Staubli VAL3: StaubliUI.pjx

--- StaubliUI.pjx ---
Parameters version=s7.7 stackSize=15000 millimeterUnit=true
Program file=Bool_Edit.pgx
Program file=BoolMess_Edit.pgx
Program file=Control_Action.pgx
Program file=Control_AxisPar.pgx
Program file=Control_BatPara.pgx
Program file=Control_BatPrt.pgx
Program file=Control_BatSpd.pgx
Program file=Control_Bottom.pgx
Program file=Control_BottomS.pgx
Program file=Control_CPreset.pgx
Program file=Control_Joint.pgx
Program file=Control_Lable.pgx
Program file=Control_Left.pgx
Program file=Control_LeftCut.pgx
Program file=Control_LeftS.pgx
Program file=Control_List.pgx
Program file=Control_List1S.pgx
Program file=Control_ListBS.pgx
Program file=Control_ListCls.pgx
Program file=Control_ListMC.pgx
Program file=Control_ListMCD.pgx
Program file=Control_ListS.pgx
Program file=Control_Loffset.pgx
Program file=Control_MCShow.pgx
Program file=Control_Mess.pgx
Program file=Control_Panel.pgx
Program file=Control_PanelB.pgx
Program file=Control_PanelD.pgx
Program file=Control_PanelMd.pgx
Program file=Control_PanelS.pgx
Program file=Control_PanelXY.pgx
Program file=Control_PanTitl.pgx
Program file=Control_Para.pgx
Program file=Control_Para1.pgx
Program file=Control_PatMove.pgx
Program file=Control_Point.pgx
Program file=Control_Preset.pgx
Program file=Control_Recipe.pgx
Program file=Control_Remote.pgx
Program file=Control_Scara.pgx
Program file=Control_Timer.pgx
Program file=Control_Traj.pgx
Program file=Control_YesNO.pgx
Program file=Float_Edit.pgx
Program file=Form_4jHome.pgx
Program file=Form_6jHome.pgx
Program file=Form_Action.pgx
Program file=Form_Bye.pgx
Program file=Form_Config.pgx
Program file=Form_LabelList.pgx
Program file=Form_Main.pgx
Program file=Form_MainS.pgx
Program file=Form_Panel.pgx
Program file=Form_Panel4P.pgx
Program file=Form_PanelBool.pgx
Program file=Form_PanelJoint.pgx
Program file=Form_PanelList.pgx
Program file=Form_PanelPoint.pgx
Program file=Form_PanelStr.pgx
Program file=Form_Patten.pgx
Program file=Form_PattenD.pgx
Program file=Form_PattenS.pgx
Program file=Form_Product.pgx
Program file=Form_ScaraRobot.pgx
Program file=Form_SelSharp.pgx
Program file=Form_SimArray.pgx
Program file=Form_Simulation.pgx
Program file=Form_Welcome.pgx
Program file=Int_Edit.pgx
Program file=Int_EditMin.pgx
Program file=Int_EditS.pgx
Program file=Key_ListBase.pgx
Program file=Key_ListMC.pgx
Program file=ReadMe.pgx
Program file=Sel_Edit.pgx
Program file=start.pgx
Program file=stop.pgx
Program file=Str_Edit.pgx
Program file=Str_SplitChar.pgx
Program file=Str_SplitComma.pgx
Data file=StaubliUI.dtx

--- Control_Action.pgx ---
public program Control_Action(num& x_nAction[] (dimensions=3), num x_nIndex, string& x_sIoName[], bool& x_bDigtal[])
  local string l_sItem[2]
  local num l_nNum
  local num l_nKey
  local num l_nData[24]
  local num l_nSelectIndex
  local bool l_bRes
  local num l_nBuff
begin
  //为LasMAN3.6 Action配置


  for l_nNum=0 to 11
    l_nData[l_nNum*2+0]=x_nAction[x_nIndex,l_nNum,0]
    l_nData[l_nNum*2+1]=x_nAction[x_nIndex,l_nNum,1]
  endFor
  l_sItem[0]="关"
  l_sItem[1]="开"

  resize(sBuff,1,24)


  call Control_BottomS("置空,清空,延时,插入,删除,,取消,确定")
  call Control_PanelXY(4,0,20,10)
  call Control_Panel("动作值")
  for l_nNum=0 to 11


    sBuff[l_nNum*2+0]=toString("",l_nNum+1)+"名称:"+x_sIoName[l_nData[l_nNum*2+0]]
    if x_bDigtal[l_nData[l_nNum*2]]
      sBuff[l_nNum*2+1]="值 : "+ l_sItem[sel(l_nData[l_nNum*2+1]==0,0,1)]
    else
      sBuff[l_nNum*2+1]="值 : "+toString(".1",l_nData[l_nNum*2+1])
    endIf

  endFor
  call Control_List(sBuff,l_nSelectIndex)


  //**********************************
  //按键响应
  while true
    l_nKey=getKey()

    switch l_nKey
      //向上
      case 261
        l_nSelectIndex=max(0,l_nSelectIndex-1)
      break

      //向下
      case 266
        l_nSelectIndex=min(l_nSelectIndex+1,23)
      break

      //编辑
      case 270
        if l_nSelectIndex%2==1
          if ! x_bDigtal[l_nData[l_nSelectIndex-1]]
            call Float_Edit(l_nData[l_nSelectIndex],nPanelLTopX+6,l_nSelectIndex+nPanelLTopY+1)
          else
            l_nData[l_nSelectIndex]=sel(l_nData[l_nSelectIndex]==1,1,0)
            call Sel_Edit(l_nData[l_nSelectIndex],nPanelLTopX+6,l_nSelectIndex+nPanelLTopY+1,l_sItem)
            l_nData[l_nSelectIndex]=sel(l_nData[l_nSelectIndex]==1,1,0)
          endIf

        else
          call Sel_Edit(l_nData[l_nSelectIndex],nPanelLTopX+7,l_nSelectIndex+nPanelLTopY+1,x_sIoName)
        endIf

      break

      case 271
        call Control_YesNO("确定设置为无IO信号吗?",l_bRes)
        if l_bRes

          l_nData[sel(l_nSelectIndex%2==0,l_nSelectIndex,l_nSelectIndex-1)]=0

        endIf

      break


      //全部置空
      case 272
        call Control_YesNO("确定全部清空吗?",l_bRes)
        if l_bRes
          for l_nNum=0 to 23
            l_nData[l_nNum]=0
          endFor


        endIf
      break


      case 273
        call Control_YesNO("确定要设置为延时吗?",l_bRes)
        if l_bRes
          l_nData[sel(l_nSelectIndex%2==0,l_nSelectIndex,l_nSelectIndex-1)]=165

        endIf
      break

      //插入
      case 274
        call Control_YesNO("确定要插入吗?",l_bRes)
        l_nBuff=roundDown(l_nSelectIndex/2)
        if l_bRes
          for l_nNum=23 to l_nBuff*2+2  step -1
            l_nData[l_nNum]=l_nData[l_nNum-2]
          endFor
          l_nData[l_nBuff*2]=l_nData[l_nBuff*2+1]=0

        endIf
      break


      //删除
      case 275
        call Control_YesNO("确定要删除吗?",l_bRes)
        l_nBuff=roundDown(l_nSelectIndex/2)
        if l_bRes
          for l_nNum=l_nBuff*2 to 21
            l_nData[l_nNum]=l_nData[l_nNum+2]
          endFor
          l_nData[23]=l_nData[22]=0

        endIf
      break





      //退出
      case 277
        cls()
        return

      break



      //取消
      case 278
        for l_nNum=0 to 11
          x_nAction[x_nIndex,l_nNum,0]= l_nData[l_nNum*2+0]
          x_nAction[x_nIndex,l_nNum,1]=l_nData[l_nNum*2+1]
        endFor
        return
      break

    endSwitch

    if l_nKey!=-1

      for l_nNum=0 to 11
        sBuff[l_nNum*2+0]=toString("",l_nNum+1)+"名称:"+x_sIoName[l_nData[l_nNum*2+0]]
        if x_bDigtal[l_nData[l_nNum*2]]
          sBuff[l_nNum*2+1]="值 : "+ l_sItem[sel(l_nData[l_nNum*2+1]==0,0,1)]
        else
          sBuff[l_nNum*2+1]="值 : "+toString(".2",l_nData[l_nNum*2+1])
        endIf

      endFor

      call Control_PanelXY(4,0,20,10)
      call Control_Panel("动作值")
      call Control_List(sBuff,l_nSelectIndex)
      call Control_BottomS("置空,清空,延时,插入,删除,,取消,确定")
    endIf


  endWhile





end

--- Control_AxisPar.pgx ---
public program Control_AxisPar(num& x_nPos, num& x_nSpeed, num& x_nPrecent, num& x_nJogSpeed, bool x_bTraj)
  local string l_sItem[6]
  local num l_nNum
  local num l_nKey
  local num l_nData[6]
  local num l_nSelectIndex
begin
  //为LasMAN3.6进行配置
  //修改点位的参数


  //通过局部变量来实现内部存储


  l_nData[0]=x_nPos
  l_nData[1]=x_nSpeed
  l_nData[2]=x_nPrecent
  l_nData[3]=x_nJogSpeed

  l_sItem[0]="位置mm   :"+toString(".3",l_nData[0])
  l_sItem[1]="速度m/min:"+toString(".3",l_nData[1])
  l_sItem[2]="比例分度 :"+toString(".3",l_nData[2])
  l_sItem[3]="点动速度 :"+toString(".3",l_nData[3])
  call Control_BottomS(",,,,,,取消,确定")

  call Control_PanelXY(8,0,17,4)
  call Control_Panel("参数")
  call Control_List(l_sItem,l_nSelectIndex)


  //按键响应
  while true
    l_nKey=getKey()

    switch l_nKey
      case 261
        l_nSelectIndex=max(0,l_nSelectIndex-1)
      break

      case 266
        if x_bTraj
          l_nSelectIndex=min(1,l_nSelectIndex+1)
        else
           l_nSelectIndex=min(3,l_nSelectIndex+1)
        endIf

      break

      case 278

        x_nPos=l_nData[0]
        x_nSpeed=l_nData[1]
        x_nPrecent=l_nData[2]
        x_nJogSpeed=l_nData[3]
        cls()
        return
      break


      case 277,255
        cls()
        return
      break



      case 270

        call Float_Edit(l_nData[l_nSelectIndex],nPanelLTopX+11,l_nSelectIndex+nPanelLTopY+1)


        l_nData[l_nSelectIndex]=max(0,l_nData[l_nSelectIndex])
        l_nData[3]=min(100,max(0,l_nData[3]))
      break

    endSwitch

    if l_nKey!=-1
      l_sItem[0]="位置mm   :"+toString(".3",l_nData[0])
      l_sItem[1]="速度m/min:"+toString(".3",l_nData[1])
      l_sItem[2]="比例分度 :"+toString(".3",l_nData[2])
      l_sItem[3]="点动速度 :"+toString(".3",l_nData[3])
      call Control_List(l_sItem,l_nSelectIndex)

    endIf






  endWhile

end

--- Control_BatPara.pgx ---
public program Control_BatPara(num x_nMax, num& x_nFrom[], num& x_nTo[], num& x_nValue[], bool& x_bEdit[])
  local string l_sItem[4]
  local num l_nNum
  local num l_nKey
  local num l_nData[6]
  local num l_nSelectIndex
  local string l_sS[5]
  local num l_nIndex
begin

  //为LasMAN3.6进行配置
  //批处理切割或者焊接点的参数
  //包括速度，加速度，blend, 工艺，动作




  x_bEdit[0]=x_bEdit[1]=x_bEdit[2]=x_bEdit[3]=x_bEdit[4]=false
  l_nData[0]=1
  l_nData[1]=x_nMax
  l_nData[2]=0
  l_nData[3]=1
  l_sS[0]="速度"
  l_sS[1]="加速度"
  l_sS[2]="Blend"
  l_sS[3]="工艺"
  l_sS[4]="动作"

  l_sItem[0]="开始序号:"+toString("",l_nData[0])
  l_sItem[1]="结束序号:"+toString("",l_nData[1])
  l_sItem[2]="选项    :"+l_sS[l_nData[2]]
  l_sItem[3]="值      :"+toString("",l_nData[3])



  call Control_BottomS(",,,,,,退出,修改")
  call Control_PanelXY(8,0,15,4)
  call Control_Panel("批处理参数")
  call Control_List(l_sItem,l_nSelectIndex)
  while true
    l_nKey=getKey()

    switch l_nKey
      case 261
        l_nSelectIndex=max(0,l_nSelectIndex-1)
      break

      case 266
        l_nSelectIndex=min(l_nSelectIndex+1,3)
      break

      case 278
        l_nIndex=round(min(max(0,l_nData[2]),4))
        x_nFrom[l_nIndex]=l_nData[0]
        x_nTo[l_nIndex]=l_nData[1]

        x_nValue[l_nIndex]=l_nData[3]
        x_bEdit[l_nIndex]=true
        popUpMsg(l_sS[l_nIndex]+"已修改")
       // cls()
        //return
      break


      case 277,255

        cls()
        //x_bEdit=false
        return
      break

      case 270
        if l_nSelectIndex==2
          call Sel_Edit(l_nData[2],nPanelLTopX+10,l_nSelectIndex+nPanelLTopY+1,l_sS)
        else
          call Float_Edit(l_nData[l_nSelectIndex],nPanelLTopX+10,l_nSelectIndex+nPanelLTopY+1)
          if l_nSelectIndex==0
            l_nData[l_nSelectIndex]=roundDown(min(l_nData[1],max(1,l_nData[l_nSelectIndex])))

          endIf
          if l_nSelectIndex==1
            l_nData[l_nSelectIndex]=roundDown(min(x_nMax,max(1,l_nData[l_nSelectIndex])))

          endIf
        endIf
      break


    endSwitch

    if l_nKey!=-1
      l_sItem[0]="开始序号:"+toString("",l_nData[0])
      l_sItem[1]="结束序号:"+toString("",l_nData[1])
      l_sItem[2]="选项    :"+l_sS[l_nData[2]]
      l_sItem[3]="值      :"+toString("",l_nData[3])

      call Control_List(l_sItem,l_nSelectIndex)

    endIf

  endWhile

end

--- Control_BatPrt.pgx ---
public program Control_BatPrt(num& x_nFrom, num& x_nTo, num& x_nPreset)
  local string l_sItem[3]
  local num l_nNum
  local num l_nKey
  local num l_nData[6]
  local num l_nSelectIndex
begin

  //为LasMAN3.6进行配置
  //批处理工艺



  l_nData[0]=x_nFrom
  l_nData[1]=x_nTo
  l_nData[2]=1
  //l_nData[3]=15
  l_sItem[0]="开始    :"+toString("",l_nData[0])
  l_sItem[1]="结束    :"+toString("",l_nData[1])
  l_sItem[2]="工艺    :"+toString("",l_nData[2])
  //  l_sItem[3]="加速度  :"+toString("",l_nData[3])



  call Control_BottomS(",,,,,,完成,修改")
  call Control_PanelXY(8,0,15,4)
  call Control_Panel("批处理工艺")
  call Control_List(l_sItem,l_nSelectIndex)
  while true
    l_nKey=getKey()

    switch l_nKey
      case 261
        l_nSelectIndex=max(0,l_nSelectIndex-1)
      break

      case 266
        l_nSelectIndex=min(l_nSelectIndex+1,2)
      break

      case 278
        x_nFrom=l_nData[0]
        x_nTo=l_nData[1]
        x_nPreset=l_nData[2]
        //   x_nAcc=l_nData[3]
        cls()
        return
      break


      case 277,255

        cls()
        return
      break

      case 270
        call Float_Edit(l_nData[l_nSelectIndex],nPanelLTopX+7,l_nSelectIndex+nPanelLTopY+1)
      break

    endSwitch

    if l_nKey!=-1
      l_nData[2]=min(max(1,l_nData[2]),50)
      l_nData[2]=round(l_nData[2])
      l_sItem[0]="开始    :"+toString("",l_nData[0])
      l_sItem[1]="结束    :"+toString("",l_nData[1])
      l_sItem[2]="工艺    :"+toString("",l_nData[2])
      // l_sItem[3]="加速度  :"+toString("",l_nData[3])
      call Control_List(l_sItem,l_nSelectIndex)

    endIf






  endWhile





end

--- Control_BatSpd.pgx ---
public program Control_BatSpd(num& x_nFrom, num& x_nTo, num& x_nSpeed, num& x_nAcc)
  local string l_sItem[4]
  local num l_nNum
  local num l_nKey
  local num l_nData[6]
  local num l_nSelectIndex
begin

  //为LasMAN3.6进行配置
  //批处理速度


  l_nData[0]=x_nFrom
  l_nData[1]=x_nTo
  l_nData[2]=100
  l_nData[3]=15
  l_sItem[0]="开始序号:"+toString("",l_nData[0])
  l_sItem[1]="结束序号:"+toString("",l_nData[1])
  l_sItem[2]="速度    :"+toString("",l_nData[2])
  l_sItem[3]="加速度  :"+toString("",l_nData[3])



  call Control_BottomS(",,,,,,取消,确定")
  call Control_PanelXY(8,0,15,4)
  call Control_Panel("批处理速度")
  call Control_List(l_sItem,l_nSelectIndex)
  while true
    l_nKey=getKey()

    switch l_nKey
      case 261
        l_nSelectIndex=max(0,l_nSelectIndex-1)
      break

      case 266
        l_nSelectIndex=min(l_nSelectIndex+1,3)
      break

      case 278
        x_nFrom=l_nData[0]
        x_nTo=l_nData[1]
        x_nSpeed=l_nData[2]
        x_nAcc=l_nData[3]
        cls()
        return
      break


      case 277,255

        cls()
        return
      break

      case 270

        call Float_Edit(l_nData[l_nSelectIndex],nPanelLTopX+7,l_nSelectIndex+nPanelLTopY+1)
      break

    endSwitch

    if l_nKey!=-1
  l_sItem[0]="开始序号:"+toString("",l_nData[0])
  l_sItem[1]="结束序号:"+toString("",l_nData[1])
  l_sItem[2]="速度    :"+toString("",l_nData[2])
  l_sItem[3]="加速度  :"+toString("",l_nData[3])
      call Control_List(l_sItem,l_nSelectIndex)

    endIf






  endWhile





end

--- Control_CPreset.pgx ---
public program Control_CPreset(num& x_nPreset[] (dimensions=2), trsf& x_trCut[], num x_nMax, num x_nIndex, trsf& x_trTrsfAxis[])
  local string l_sItem[6]
  local num l_nNum
  local num l_nKey
  local num l_nData[5]
  local num l_nIndex
  local num l_nBuff
  local bool l_bFirst
  local bool l_bEdit
begin

  //为LasMAN3.6进行定制
  //修改工艺参数


  //  //把传入参数临时存储
  //  l_nIndex=x_trCut[x_nIndex].x
  //  for l_nNum=0 to 4
  //    l_nData[l_nNum]=x_nPreset[l_nIndex,l_nNum]
  //  endFor
  //
  //  //界面初始化
  //      l_sItem[0]="工艺号  :"+toString("",l_nIndex)
  //      l_sItem[1]="激光功率  :"+toString("",l_nData[0])
  //      l_sItem[2]="气体压力  :"+toString("",l_nData[1])
  //      l_sItem[3]="占空比频率:"+toString("",l_nData[2])
  //      l_sItem[4]="激光占空比:"+toString("",l_nData[3])
  //      l_sItem[5]="随动高度  :"+toString("",l_nData[4])
  //      call Control_List(l_sItem,l_nBuff)


  //2015.03.10
  //天虹激光进行修改过




  l_nIndex=x_trCut[x_nIndex].x
  call Control_BottomS(",,,,,,退出,应用")
  call Control_PanelXY(8,0,15,6)
  call Control_Panel(toString("",x_nIndex)+":工艺值")
  call Control_List(l_sItem,l_nBuff)
  //按键响应



  //
  if x_trCut[x_nIndex].x==0

    l_nData[0]=x_trTrsfAxis[x_nIndex].rx
    l_nData[1]=x_trTrsfAxis[x_nIndex].ry

  endIf


  while true
    l_nKey=getKey()

    switch l_nKey
      //上
      case 261
        if l_bEdit
          l_nData[0]=max(0,l_nData[0]-1)
        else
          l_nIndex=max(0,l_nIndex-1)
        endIf
        //l_nSelectIndex=max(0,l_nSelectIndex-1)
      break


      //下
      case 266
        if l_bEdit
          l_nData[0]=min(100,l_nData[0]+1)
        else
          l_nIndex=min(50,l_nIndex+1)
        endIf
        // l_nSelectIndex=min(l_nSelectIndex+1,5)
      break



      //<-  向左修改点序号
      case 264

        if l_bEdit
          l_nData[1]=max(0,l_nData[1]-1)
        else
          x_nIndex=max(0,x_nIndex-1)
          l_nIndex=x_trCut[x_nIndex].x
          if x_trCut[x_nIndex].x==0

            l_nData[0]=x_trTrsfAxis[x_nIndex].rx
            l_nData[1]=x_trTrsfAxis[x_nIndex].ry

          endIf
        endIf
      break


      //-> 改点序号
      case 268
        if l_bEdit
          l_nData[1]=min(100,l_nData[1]+1)
        else
          x_nIndex=min(x_nMax-1,x_nIndex+1)
          l_nIndex=x_trCut[x_nIndex].x
          if x_trCut[x_nIndex].x==0

            l_nData[0]=x_trTrsfAxis[x_nIndex].rx
            l_nData[1]=x_trTrsfAxis[x_nIndex].ry

          endIf
        endIf
      break



      case 270
        if l_nIndex==0

          l_bEdit=!l_bEdit

        endIf

      break


      //应用
      case 278
        //        for l_nNum=0 to 4
        //          x_nPreset[x_nIndex,l_nNum]=min(max(l_nData[l_nNum],0),100)
        //      x.x=l_nIndex
        x_trCut[x_nIndex].x=l_nIndex
        //   return
      //  l_nIndex=x_trCut[x_nIndex].x
        if l_nIndex==0
          x_trTrsfAxis[x_nIndex].rx=l_nData[0]
          x_trTrsfAxis[x_nIndex].ry=l_nData[1]

        endIf
      break



      case 277
        return
      break

      //      case 270
      //        call Float_Edit(l_nData[l_nSelectIndex],nPanelLTopX+12,l_nSelectIndex+nPanelLTopY+1)
      //        l_nData[l_nSelectIndex]=min(max(l_nData[l_nSelectIndex],0),100)
      //      break

    endSwitch

    if l_nIndex!=0
      l_bEdit=false
    endIf


    if l_nKey!=-1 or !l_bFirst
      l_bFirst=true

      call Control_PanTitl(toString("",x_nIndex+1)+"点:工艺值")

      if l_nIndex!=0
        for l_nNum=0 to 4
          l_nData[l_nNum]=x_nPreset[l_nIndex,l_nNum]
        endFor
        //      for l_nNum=0 to 4
        //        l_nData[l_nNum]=x_nPreset[l_nIndex,l_nNum]
        //      endFor
        l_sItem[0]="工艺号    :"+toString("",l_nIndex)
        l_sItem[1]="激光功率  :"+toString("",l_nData[0])
        l_sItem[2]="气体压力  :"+toString("",l_nData[1])
        l_sItem[3]="占空比频率:"+toString("",l_nData[2])
        l_sItem[4]="激光占空比:"+toString("",l_nData[3])
        l_sItem[5]="随动高度  :"+toString("",l_nData[4])

      else

        l_sItem[0]="工艺号    :"+toString("",l_nIndex)
        l_sItem[1]="激光功率  :"+toString("",l_nData[0])
        l_sItem[2]="激光占空比:"+toString("",l_nData[1])
        if l_bEdit
          l_sItem[4]="按上下修改功率 "
          l_sItem[5]="按左右修改占空比"
        else
          l_sItem[4]="按Enter修改    "
          l_sItem[5]="               "
        endIf

        l_sItem[3]="               "

      endIf





      call Control_List(l_sItem,l_nBuff)





    endIf







  endWhile





end

--- Control_List.pgx ---
public program Control_List(string& x_sItemName[], num& x_nSelectItem)
  local num l_nIndex
  local bool l_bRes
  local num l_nFrist
  local num l_nNum
  local bool l_bBlack
  local bool l_bBlank
  local num l_nCount
  local string l_sBuff
begin
  //说明：
  //函数功能：在划定的框内，把选中项给显示出来
  //l_nFirst  在列表中第一个显示的项的序号
  //x_nSelectItem  被选中的项的序号
  //l_nCount 合法列表项的项总数，如何数组中间为空，则可能被截断


  //1.参数初始化
  l_nFrist=0
  l_nCount=0

  //2.参数合法化判断，得到合法项的总数
  for l_nIndex=0 to size(x_sItemName)-1
    if x_sItemName[l_nIndex]==""
      l_nIndex=size(x_sItemName)
    else
      l_nCount=l_nCount+1
    endIf
  endFor

  //3.如果选中项大于列表长度
  x_nSelectItem=min(max(0,x_nSelectItem),l_nCount-1)
  if x_nSelectItem>=nPanelLengthY
    l_nFrist=x_nSelectItem-nPanelLengthY+1
  endIf


  //4.把列表给画出来
  for l_nIndex=0 to min(nPanelLengthY-1,l_nCount-l_nFrist-1)
    gotoxy(nPanelLTopX+1,nPanelLTopY+l_nIndex+1)
    setTextMode(sel(l_nIndex+l_nFrist==x_nSelectItem,1,0))
    //l_nNum=max(nPanelWidthX-getDisplayLen(x_sItemName[l_nIndex+l_nFrist])+len(x_sItemName[l_nIndex+l_nFrist]),nPanelWidthX)
   l_sBuff=left(x_sItemName[l_nIndex+l_nFrist]+"                                  ",nPanelWidthX)
   while getDisplayLen(l_sBuff)>nPanelWidthX
  l_sBuff=left(l_sBuff,len(l_sBuff)-1)
  endWhile
  put(l_sBuff)
//   left(x_sItemName[x_sItemName[l_nIndex+l_nFrist]],nPanelWidthX-)
//    put(left(x_sItemName[l_nIndex+l_nFrist]+"                            ",l_nNum))





  endFor


  //5.对剩下的进行补空
  setTextMode(0)
  while l_nIndex< nPanelLengthY
    gotoxy(nPanelLTopX+1,nPanelLTopY+l_nIndex+1)
    put(left("                               ",nPanelWidthX))
    l_nIndex=l_nIndex+1
  endWhile


end

--- Control_Loffset.pgx ---
public program Control_Loffset(num& x_nFrom, num& x_nTo)
  local string l_sItem[2]
  local num l_nNum
  local num l_nKey
  local num l_nData[6]
  local num l_nSelectIndex
begin

  //为LasMAN3.6配置
  //局部偏差
l_nData[0]=x_nFrom
l_nData[1]=x_nTo

  l_sItem[0]="开始    :"+toString("",l_nData[0])
  l_sItem[1]="停止    :"+toString("",l_nData[1])
  call Control_BottomS(",,,,,,取消,确定")
  call Control_PanelXY(8,0,15,6)
  call Control_Panel("局部偏差值")
  call Control_List(l_sItem,l_nSelectIndex)
  while true
    l_nKey=getKey()

    switch l_nKey
      case 261
        l_nSelectIndex=max(0,l_nSelectIndex-1)
      break

      case 266
        l_nSelectIndex=min(l_nSelectIndex+1,1)
      break

      case 278
          x_nFrom=l_nData[0]
          x_nTo=l_nData[1]
         cls()
        return
      break


      case 277,255

        cls()
        return
      break

      case 270
        call Float_Edit(l_nData[l_nSelectIndex],nPanelLTopX+7,l_nSelectIndex+nPanelLTopY+1)
      break

    endSwitch

    if l_nKey!=-1
  l_sItem[0]="开始    :"+toString("",l_nData[0])
  l_sItem[1]="停止    :"+toString("",l_nData[1])
      call Control_List(l_sItem,l_nSelectIndex)

    endIf






  endWhile





end

--- Control_MCShow.pgx ---
public program Control_MCShow(num x_nIndex, num x_nMoveType)
  local string l_sS[3]
begin

  //LasMAN3.6
  //为圆弧进行配置

  if x_nMoveType>2 or x_nMoveType<1
    return
  endIf
  l_sS[0]=toString("",x_nIndex+1)+"."+"MoveC "
  l_sS[1]=toString("",1)+" "
  l_sS[2]=left(" "+toString("",2)+"       ",nPanelWidthX-len(l_sS[0])-len(l_sS[1]))
  setTextMode(0)
  gotoxy(nPanelLTopX+1,min(nPanelLengthY,x_nIndex+1))
  put(l_sS[0])
  setTextMode(sel(x_nMoveType==1,1,0))
  put(l_sS[1])
  setTextMode(sel(x_nMoveType==1,0,1))
  put(l_sS[2])


  setTextMode(0)

end

--- Control_Para.pgx ---
public program Control_Para(trsf& x_trTrsf[], bool& x_bRes[], bool x_bCut, num x_nTrajType, num x_nId, trsf& x_trExtAxis[])
  local string l_sItem[8]
  local num l_nNum
  local num l_nKey
  local num l_nData[8]
  local num l_nSelectIndex
  local bool l_bFrist
  local num l_nFid
begin
  //为LasMAN3.6进行配置
  //修改点位的参数


  l_nFid=x_nId

  call Control_BottomS(",,,,,,退出,修改")
  if x_bCut
    if x_nTrajType!=10 and x_nTrajType!=20 and x_nTrajType!=9
      call Control_PanelXY(8,0,18,5)
    else
      if x_nTrajType==10
        call Control_PanelXY(8,0,18,6)
      else
        call Control_PanelXY(8,0,18,8)
      endIf
    endIf
  else
    if x_nTrajType==20
      call Control_PanelXY(8,0,17,5)
    else
      call Control_PanelXY(8,0,17,3)
    endIf
  endIf

  call Control_Panel("参数")
  call Control_List(l_sItem,l_nSelectIndex)


  //按键响应
  while true
    l_nKey=getKey()

    switch l_nKey
      case 261
        l_nSelectIndex=max(0,l_nSelectIndex-1)
      break

      case 264
        x_nId=max(0,x_nId-1)
      break


      case 268
        x_nId=min(size(x_trTrsf)-1,x_nId+1)
      break

      case 266
        if x_bCut
          if x_nTrajType==10
            l_nSelectIndex=min(l_nSelectIndex+1,5)
          else
            if x_nTrajType==20
              l_nSelectIndex=min(l_nSelectIndex+1,7)
            else
              l_nSelectIndex=min(l_nSelectIndex+1,4)
            endIf
          endIf
        else
          if x_nTrajType==20
            l_nSelectIndex=min(l_nSelectIndex+1,4)
          else
            l_nSelectIndex=min(l_nSelectIndex+1,2)
          endIf

        endIf
      break

      case 278
        if l_nFid!=x_nId and x_bRes[x_nId]!=(l_nNum==1)
          popUpMsg("运动类型需在当前位置点修改")
        else
          x_trTrsf[x_nId].x=l_nData[3]
          x_trTrsf[x_nId].y=l_nData[4]
          x_trTrsf[x_nId].z=l_nData[0]
          x_trTrsf[x_nId].rx=l_nData[1]

          x_trTrsf[x_nId].ry=l_nData[2]
          x_trTrsf[x_nId].rz=l_nData[5]
          if x_bCut
            x_trExtAxis[x_nId].x=l_nData[6]
            x_trExtAxis[x_nId].y=l_nData[7]
          else
            x_trExtAxis[x_nId].x=l_nData[3]
            x_trExtAxis[x_nId].y=l_nData[4]
          endIf
          x_bRes[x_nId]=(l_nNum==1)
          gotoxy(0,13)
          put(toString("",x_nId+1)+":参数已修改")
        endIf
      break


      case 277,255
        cls()
        return
      break



      case 270
        if (l_nSelectIndex==2 and !x_bCut) or (l_nSelectIndex==5 and x_bCut)
          call Sel_Edit(l_nNum,nPanelLTopX+11,l_nSelectIndex+nPanelLTopY+1,sData)

        else
          call Float_Edit(l_nData[l_nSelectIndex],nPanelLTopX+11,l_nSelectIndex+nPanelLTopY+1)
        endIf
      break

    endSwitch

    if l_nKey!=-1 or !l_bFrist
      //      if x_bCut
      //
      //        sData[0]="直线"
      //        sData[1]="圆弧"
      //        l_sItem[0]="速度(mm/s:"+toString(".3",l_nData[0])
      //        l_sItem[1]="加速度(%):"+toString(".3",l_nData[1])
      //        l_sItem[2]="BLend(mm):"+toString(".3",l_nData[2])
      //        l_sItem[3]="工艺     :"+toString(".3",l_nData[3])
      //        l_sItem[4]="动作     :"+toString(".3",l_nData[4])
      //        l_sItem[5]="圆弧/直线:"+sData[l_nNum]
      //
      //      else
      //        sData[0]="MoveJ"
      //        sData[1]="MoveL"
      //        l_sItem[0]="速度(mm/s:"+toString(".3",l_nData[0])
      //        l_sItem[1]="加速度(%):"+toString(".3",l_nData[1])
      //        l_sItem[2]="关节/直线:"+sData[l_nNum]
      //
      //      endIf

      //通过局部变量来实现内部存储
      if !l_bFrist or l_nKey==264  or l_nKey==268
        l_bFrist=true
        if x_bCut
          l_nData[3]=x_trTrsf[x_nId].x
          l_nData[4]=x_trTrsf[x_nId].y
          l_nData[0]=x_trTrsf[x_nId].z
          l_nData[1]=x_trTrsf[x_nId].rx

          l_nData[2]=x_trTrsf[x_nId].ry
          l_nData[5]=x_trTrsf[x_nId].rz


          l_nData[6]=x_trExtAxis[x_nId].x
          l_nData[7]=x_trExtAxis[x_nId].y
        else
          l_nData[0]=x_trTrsf[x_nId].z
          l_nData[1]=x_trTrsf[x_nId].rx

          l_nData[3]=x_trExtAxis[x_nId].x
          l_nData[4]=x_trExtAxis[x_nId].y


        endIf

        l_nNum=sel(x_bRes[x_nId],1,0)

        //界面初始化
        resize(sData,1,2)
        call Control_PanTitl(toString("",x_nId+1)+":参数")
      endIf
      if x_bCut

        sData[0]="直线"
        sData[1]="圆弧"
        l_sItem[0]="速度(mm/s:"+toString(".3",l_nData[0])
        l_sItem[1]="加速度(%):"+toString(".3",l_nData[1])
        l_sItem[2]="BLend(mm):"+toString(".3",l_nData[2])
        l_sItem[3]="工艺     :"+toString(".3",l_nData[3])
        l_sItem[4]="动作     :"+toString(".3",l_nData[4])
        l_sItem[5]="圆弧/直线:"+sData[l_nNum]
        l_sItem[6]="同步七轴 :"+toString(".3",l_nData[6])
        l_sItem[7]="同步八轴 :"+toString(".3",l_nData[7])

      else
        sData[0]="MoveJ"
        sData[1]="MoveL"
        l_sItem[0]="速度(mm/s:"+toString(".3",l_nData[0])
        l_sItem[1]="加速度(%):"+toString(".3",l_nData[1])
        l_sItem[2]="关节/直线:"+sData[l_nNum]
        l_sItem[3]="同步七轴 :"+toString(".3",l_nData[3])
        l_sItem[4]="同步八轴 :"+toString(".3",l_nData[4])

      endIf



      call Control_List(l_sItem,l_nSelectIndex)

    endIf






  endWhile

end

--- Control_Para1.pgx ---
public program Control_Para1(trsf& x_trTrsf, bool& x_bRes, bool x_bCut, num x_nType)
  local string l_sItem[6]
  local num l_nNum
  local num l_nKey
  local num l_nData[6]
  local num l_nSelectIndex
begin
  //为LasMAN3.6进行配置
  //修改点位的参数


  //通过局部变量来实现内部存储
  l_nData[3]=x_trTrsf.x
  l_nData[4]=x_trTrsf.y
  l_nData[0]=x_trTrsf.z
  l_nData[1]=x_trTrsf.rx

  l_nData[2]=x_trTrsf.ry
  l_nData[5]=x_trTrsf.rz
  l_nNum=sel(x_bRes,1,0)

  //界面初始化
  resize(sData,1,2)
  if x_bCut

    sData[0]="直线"
    sData[1]="圆弧"
    l_sItem[0]="速度(mm/s:"+toString(".3",l_nData[0])
    l_sItem[1]="加速度(%):"+toString(".3",l_nData[1])
    l_sItem[2]="BLend(mm):"+toString(".3",l_nData[2])
    l_sItem[3]="工艺     :"+toString(".3",l_nData[3])
    l_sItem[4]="动作     :"+toString(".3",l_nData[4])
    l_sItem[5]="圆弧/直线:"+sData[l_nNum]

  else
    sData[0]="MoveJ"
    sData[1]="MoveL"
    l_sItem[0]="速度(mm/s:"+toString(".3",l_nData[0])
    l_sItem[1]="加速度(%):"+toString(".3",l_nData[1])
    l_sItem[2]="关节/直线:"+sData[l_nNum]

  endIf

  call Control_BottomS(",,,,,,取消,确定")
  if x_bCut
    if x_nType!=10
      call Control_PanelXY(8,0,18,5)
    else
      call Control_PanelXY(8,0,18,6)
    endIf
  else
    call Control_PanelXY(8,0,17,3)
  endIf
  call Control_Panel("参数")
  call Control_List(l_sItem,l_nSelectIndex)


  //按键响应
  while true
    l_nKey=getKey()

    switch l_nKey
      case 261
        l_nSelectIndex=max(0,l_nSelectIndex-1)
      break

      case 266
        if x_bCut
          if x_nType==10
            l_nSelectIndex=min(l_nSelectIndex+1,5)
          else
            l_nSelectIndex=min(l_nSelectIndex+1,4)
          endIf
        else
          l_nSelectIndex=min(l_nSelectIndex+1,2)
        endIf
      break

      case 278
        x_trTrsf.x=l_nData[3]
        x_trTrsf.y=l_nData[4]
        x_trTrsf.z=l_nData[0]
        x_trTrsf.rx=l_nData[1]

        x_trTrsf.ry=l_nData[2]
        x_trTrsf.rz=l_nData[5]
        x_bRes=(l_nNum==1)
        cls()
        return
      break


      case 277,255
        cls()
        return
      break



      case 270
        if (l_nSelectIndex==2 and !x_bCut) or (l_nSelectIndex==5 and x_bCut)
          call Sel_Edit(l_nNum,nPanelLTopX+11,l_nSelectIndex+nPanelLTopY+1,sData)

        else
          call Float_Edit(l_nData[l_nSelectIndex],nPanelLTopX+11,l_nSelectIndex+nPanelLTopY+1)
        endIf
      break

    endSwitch

    if l_nKey!=-1
      if x_bCut

        sData[0]="直线"
        sData[1]="圆弧"
        l_sItem[0]="速度(mm/s:"+toString(".3",l_nData[0])
        l_sItem[1]="加速度(%):"+toString(".3",l_nData[1])
        l_sItem[2]="BLend(mm):"+toString(".3",l_nData[2])
        l_sItem[3]="工艺     :"+toString(".3",l_nData[3])
        l_sItem[4]="动作     :"+toString(".3",l_nData[4])
        l_sItem[5]="圆弧/直线:"+sData[l_nNum]

      else
        sData[0]="MoveJ"
        sData[1]="MoveL"
        l_sItem[0]="速度(mm/s:"+toString(".3",l_nData[0])
        l_sItem[1]="加速度(%):"+toString(".3",l_nData[1])
        l_sItem[2]="关节/直线:"+sData[l_nNum]

      endIf
      call Control_List(l_sItem,l_nSelectIndex)

    endIf






  endWhile

end

--- Control_PatMove.pgx ---
public program Control_PatMove(num& x_nStart, num& x_nEnd)
  local string l_sItem[6]
  local num l_nNum
  local num l_nKey
  local num l_nData[6]
  local num l_nSelectIndex
begin
  //为LasMAN3.6进行配置
  //中途进行模拟点

  l_nData[0]=x_nStart
  l_nData[1]=x_nEnd


  l_sItem[0]="开始模拟点:"+toString(".3",l_nData[0])
  l_sItem[1]="结束模拟点:"+toString(".3",l_nData[1])


  call Control_BottomS(",,,,,,,确定")
  call Control_PanelXY(8,0,15,2)
  call Control_Panel("切割点局部模拟")
  call Control_List(l_sItem,l_nSelectIndex)
  while true
    l_nKey=getKey()

    switch l_nKey
      case 261
        l_nSelectIndex=max(0,l_nSelectIndex-1)
      break

      case 266
        l_nSelectIndex=min(l_nSelectIndex+1,1)
      break

      case 278
        x_nStart=l_nData[0]
        x_nEnd=l_nData[1]
        cls()
        return
      break


      //      case 277,255
      //
      //        cls()
      //        return
      //      break

      case 270
        call Float_Edit(l_nData[l_nSelectIndex],nPanelLTopX+12,l_nSelectIndex+nPanelLTopY+1)
      break

    endSwitch

    if l_nKey!=-1
      l_sItem[0]="开始模拟点:"+toString(".3",l_nData[0])
      l_sItem[1]="结束模拟点:"+toString(".3",l_nData[1])

      call Control_List(l_sItem,l_nSelectIndex)

    endIf






  endWhile





end

--- Control_Preset.pgx ---
public program Control_Preset(num& x_nPreset[] (dimensions=2), num x_nIndex)
  local string l_sItem[5]
  local num l_nNum
  local num l_nKey
  local num l_nData[5]
  local num l_nSelectIndex
begin

  //为LasMAN3.6进行定制
  //修改工艺参数


  //把传入参数临时存储
  for l_nNum=0 to 4
    l_nData[l_nNum]=x_nPreset[x_nIndex,l_nNum]
  endFor

  //界面初始化
  l_sItem[0]="激光功率  :"+toString("",l_nData[0])
  l_sItem[1]="气体压力  :"+toString("",l_nData[1])
  l_sItem[2]="占空比频率:"+toString("",l_nData[2])
  l_sItem[3]="激光占空比:"+toString("",l_nData[3])
  l_sItem[4]="随动高度  :"+toString("",l_nData[4])

  call Control_BottomS(",,,,,,取消,确定")
  call Control_PanelXY(8,0,15,5)
  call Control_Panel("工艺值")
  call Control_List(l_sItem,l_nSelectIndex)
  //按键响应
  while true
    l_nKey=getKey()

    switch l_nKey
      case 261
        l_nSelectIndex=max(0,l_nSelectIndex-1)
      break

      case 266
        l_nSelectIndex=min(l_nSelectIndex+1,5)
      break

      case 278
        for l_nNum=0 to 4
          x_nPreset[x_nIndex,l_nNum]=min(max(l_nData[l_nNum],0),100)
        endFor
        return
      break


      case 277
        return
      break

      case 270
        call Float_Edit(l_nData[l_nSelectIndex],nPanelLTopX+12,l_nSelectIndex+nPanelLTopY+1)
        l_nData[l_nSelectIndex]=min(max(l_nData[l_nSelectIndex],0),100)
      break

    endSwitch

    if l_nKey!=-1

      l_sItem[0]="激光功率  :"+toString("",l_nData[0])
      l_sItem[1]="气体压力  :"+toString("",l_nData[1])
      l_sItem[2]="占空比频率:"+toString("",l_nData[2])
      l_sItem[3]="激光占空比:"+toString("",l_nData[3])
      l_sItem[4]="随动高度  :"+toString("",l_nData[4])
      call Control_List(l_sItem,l_nSelectIndex)

    endIf






  endWhile





end

--- Control_Remote.pgx ---
public program Control_Remote(num& x_nMode, num& x_nCycleCount)
  local string l_sItem[2]
  local num l_nNum
  local num l_nKey
  local num l_nData[2]
  local num l_nSelectIndex
  local string l_sSMess[6]
begin

  //为LasMAN3.6进行配置
  //主要是远程选择界面



  l_nData[0]=max(round(x_nMode),0)
  l_nData[1]=max(round(x_nCycleCount),0)

  l_sSMess[0]="按钮触发单工位"
  l_sSMess[1]="按钮触发单周期"
  l_sSMess[2]="按钮触发多周期"
  l_sSMess[3]="无需按钮触发"
  l_sSMess[4]="按钮触发排队"
  l_sSMess[5]="用户自定义触发"


  l_sItem[0]="生产模式:"+l_sSMess[l_nData[0]]
  l_sItem[1]="周期次数:"+toString("",l_nData[1])


  call Control_BottomS(",,,,,,取消,确定")
  call Control_PanelXY(8,0,25,2)
  call Control_ListCls()
  call Control_Panel("生产配置")
  call Control_List(l_sItem,l_nSelectIndex)
  while true
    l_nKey=getKey()

    switch l_nKey
      case 261
        l_nSelectIndex=max(0,l_nSelectIndex-1)
        //        l_nSelectIndex=l_nSelectIndex-1
        //        if l_nSelectIndex<=-1
        //          l_nSelectIndex=5
        //        endIf

      break

      case 266
        l_nSelectIndex=min(l_nSelectIndex+1,1)
        //       l_nSelectIndex=l_nSelectIndex+1
        //       if l_nSelectIndex>=6
        //        l_nSelectIndex=0
        //      endIf
      break

      case 278
        x_nMode=l_nData[0]
        x_nCycleCount=l_nData[1]

        return
      break


      case 277
        return
      break

      case 270
        if l_nSelectIndex==0
          call Sel_Edit(l_nData[0],nPanelLTopX+10,nPanelLTopY+1,l_sSMess)
        else
          call Float_Edit(l_nData[1],nPanelLTopX+10,nPanelLTopY+2)

        endIf



        l_nData[l_nSelectIndex]=max(round(l_nData[l_nSelectIndex]),0)
      break

    endSwitch

    if l_nKey!=-1
      l_sItem[0]="生产模式:"+l_sSMess[l_nData[0]]
      l_sItem[1]="周期次数:"+toString("",l_nData[1])
      call Control_List(l_sItem,l_nSelectIndex)

    endIf






  endWhile





end

--- Control_Traj.pgx ---
public program Control_Traj(trsf& x_trFrame, trsf& x_trOffset, trsf& x_trArray, trsf& x_trDownLead, trsf& x_trWorkPlace, bool& x_bInerCut, num& x_nDelay[], num& x_nLength[], bool x_bWeld)
  local num l_nSelectIndex
  local num l_nData[40]
  local num l_nKey
  local num l_nNum
  local bool l_bFirst
begin
  //修改点位的 joint


  // x_trDownLead.rz只能是大于10
  //圆弧度
  l_nData[10]=x_trFrame.x
  l_nData[11]=x_trFrame.y
  l_nData[12]=x_trFrame.z
  l_nData[13]=x_trFrame.rx
  l_nData[14]=x_trFrame.ry
  l_nData[15]=x_trFrame.rz

  l_nData[16]=x_trOffset.x
  l_nData[17]=x_trOffset.y
  l_nData[18]=x_trOffset.z
  l_nData[19]=x_trOffset.rx
  l_nData[20]=x_trOffset.ry
  l_nData[21]=x_trOffset.rz

  l_nData[2]=x_trArray.x
  l_nData[3]=x_trArray.y
  l_nData[4]=x_trArray.z
  l_nData[5]=x_trArray.rx

  l_nData[6]=x_trDownLead.x
  l_nData[7]=x_trDownLead.y
  l_nData[8]=x_trDownLead.z
  l_nData[9]=x_trDownLead.rx

  l_nData[0]=x_trDownLead.ry
  //圆弧度
  l_nData[1]=x_trDownLead.rz*10

  l_nData[22]=x_trWorkPlace.x
  l_nData[23]=x_trWorkPlace.y



  l_nData[24]=sel(x_bInerCut,0,1)
  l_nData[25]=x_nDelay[0]
  l_nData[26]=x_nDelay[1]
  l_nData[27]=x_nLength[0]
  l_nData[28]=x_nLength[1]
  l_nData[29]=x_trWorkPlace.ry
  l_nData[30]=x_trWorkPlace.rz

  l_nData[31]=x_trWorkPlace.z
  l_nData[32]=x_trWorkPlace.rx

  //2016.01.13
  //为焊接添加Z轴方向的阵列
  l_nData[33]=x_trArray.ry
  l_nData[34]=x_trArray.rz


  //  resize(sData,1,3)
  //  sData[0]="无"
  //  sData[1]="直线"
  //  sData[2]="圆弧"
  //
  //  resize(sBuff,1,31)
  //  sBuff[0]="圆直径    :"+toString(".3",l_nData[0])
  //  sBuff[1]="圆弧度(焊):"+toString(".3",l_nData[1])
  //
  //  sBuff[2]="X方向个数 :"+toString("",l_nData[2])
  //  sBuff[3]="X方向距离 :"+toString(".3",l_nData[3])
  //  sBuff[4]="Y方向个数 :"+toString("",l_nData[4])
  //  sBuff[5]="Y方向距离 :"+toString(".3",l_nData[5])
  //
  //  sBuff[6]="引入类型  :"+sData[l_nData[6]]
  //  sBuff[7]="引入比例  :"+toString(".3",l_nData[7])
  //  sBuff[8]="引出类型  :"+sData[l_nData[8]]
  //  sBuff[9]="引出比例  :"+toString(".3",l_nData[9])
  //
  //
  //
  //  sBuff[10]="坐标系X   :"+toString(".3",l_nData[10])
  //  sBuff[11]="坐标系Y   :"+toString(".3",l_nData[11])
  //  sBuff[12]="坐标系Z   :"+toString(".3",l_nData[12])
  //  sBuff[13]="坐标系RX  :"+toString(".3",l_nData[13])
  //  sBuff[14]="坐标系RY  :"+toString(".3",l_nData[14])
  //  sBuff[15]="坐标系RZ  :"+toString(".3",l_nData[15])
  //
  //
  //  sBuff[16]="路径偏差X :"+toString(".3",l_nData[16])
  //  sBuff[17]="路径偏差Y :"+toString(".3",l_nData[17])
  //  sBuff[18]="路径偏差Z :"+toString(".3",l_nData[18])
  //  sBuff[19]="路径偏差RX:"+toString(".3",l_nData[19])
  //  sBuff[20]="路径偏差RY:"+toString(".3",l_nData[20])
  //  sBuff[21]="路径偏差RZ:"+toString(".3",l_nData[21])
  //
  //
  //  sBuff[22]="七轴距离  :"+toString(".3",l_nData[22])
  //  sBuff[23]="七轴速度  :"+toString(".3",l_nData[23])
  //  sBuff[25]="激光开延时:"+toString(".3",l_nData[25])
  //  sBuff[26]="激光关延时:"+toString(".3",l_nData[26])
  //  sBuff[27]="边长1     :"+toString(".3",l_nData[27])
  //  sBuff[28]="边长2     :"+toString(".3",l_nData[28])
  //  sBuff[29]="收弧时间  :"+toString(".3",l_nData[29])
  //  resize(sData,1,2)
  //  if !x_bWeld
  //    sData[0]="内切"
  //    sData[1]="外切"
  //    sBuff[24]="类型      :"+sData[l_nData[24]]
  //  else
  //    sData[0]="开"
  //    sData[1]="关"
  //    sBuff[24]="使用动作  :"+sData[l_nData[24]]
  //
  //  endIf
  //
  //  sBuff[24]="类型      :"+sData[l_nData[24]]
  //  if !x_bWeld
  //    sBuff[30]="穿孔工艺:"+toString(".3",l_nData[30])
  //  else
  //    sBuff[30]="激光程序号:"+toString(".3",l_nData[30])
  //  endIf


  call Control_BottomS(",,,,,,取消,确定")
  call Control_PanelXY(8,0,17,11)
  call Control_Panel("路径参数")
  call Control_List(sBuff,l_nSelectIndex)
  while true
    l_nKey=getKey()

    switch l_nKey
      case 261
        //        l_nSelectIndex=max(0,l_nSelectIndex-1)

        l_nSelectIndex=l_nSelectIndex-1
        if l_nSelectIndex<=-1
          l_nSelectIndex=size(sBuff)-1
        endIf

      break

      case 266
        l_nSelectIndex=l_nSelectIndex+1
        if l_nSelectIndex>=size(sBuff)
          l_nSelectIndex=0
        endIf
        //l_nSelectIndex=min(l_nSelectIndex+1,size(sBuff)-1)
      break

      case 278
        x_trFrame.x=l_nData[10]
        x_trFrame.y =l_nData[11]
        x_trFrame.z=l_nData[12]
        x_trFrame.rx =l_nData[13]
        x_trFrame.ry =l_nData[14]
        x_trFrame.rz =l_nData[15]

        x_trOffset.x=l_nData[16]
        x_trOffset.y =l_nData[17]
        x_trOffset.z =l_nData[18]
        x_trOffset.rx =l_nData[19]
        x_trOffset.ry =l_nData[20]
        x_trOffset.rz =l_nData[21]

        x_trArray.x=l_nData[2]
        x_trArray.y= l_nData[3]
        x_trArray.z= l_nData[4]
        x_trArray.rx= l_nData[5]

        x_trDownLead.x= l_nData[6]
        x_trDownLead.y= l_nData[7]
        x_trDownLead.z= l_nData[8]
        x_trDownLead.rx= l_nData[9]
        x_trDownLead.ry= l_nData[0]
        x_trDownLead.rz= l_nData[1]/10

        x_trWorkPlace.x= l_nData[22]
        x_trWorkPlace.y= l_nData[23]
        x_bInerCut=l_nData[24]==0
        x_nDelay[0]=l_nData[25]
        x_nDelay[1]=l_nData[26]
        x_nLength[0]=l_nData[27]
        x_nLength[1]=l_nData[28]
        x_trWorkPlace.ry=l_nData[29]

        //2016.01.13
        //为焊接添加Z轴方向的阵列
        x_trArray.ry= l_nData[33]
        x_trArray.rz= l_nData[34]

        //2015.02.02
        //为同步轴修改
        if l_nData[30]!=-1
          x_trWorkPlace.rz=min(50,max(l_nData[30],1))
        else
          x_trWorkPlace.rz=-1
        endIf
        x_trWorkPlace.z= l_nData[31]
        x_trWorkPlace.rx= l_nData[32]
        cls()
        return
      break


      case 277,255
        cls()
        return
      break

      case 270
        switch l_nSelectIndex
          //          case 4
          //            call Int_Edit(l_nData[l_nSelectIndex],nPanelLTopX+12,sel(l_nSelectIndex>=10,10,l_nSelectIndex)+nPanelLTopY+1)
          //          break

          case 30
            call Int_EditMin(l_nData[l_nSelectIndex],nPanelLTopX+12,sel(l_nSelectIndex>=10,10,l_nSelectIndex)+nPanelLTopY+1,"",-1)
          break

          case 0,1,2,3,4,5,7,9,10,11,12,13,14,15,16,17,18,19,20,21,22,23,25,26,27,28,29,31,32,33,34
            call Float_Edit(l_nData[l_nSelectIndex],nPanelLTopX+12,sel(l_nSelectIndex>=10,10,l_nSelectIndex)+nPanelLTopY+1)
          break
          case 6,8,24
            if l_nSelectIndex>9
              resize(sData,1,2)
              if !x_bWeld
                sData[0]="内切"
                sData[1]="外切"
              else
                sData[0]="开"
                sData[1]="关"
              endIf
            else
              resize(sData,1,3)
              sData[0]="无"
              sData[1]="直线"
              sData[2]="圆弧"
            endIf
            call Sel_Edit(l_nData[l_nSelectIndex],nPanelLTopX+12,sel(l_nSelectIndex>=10,10,l_nSelectIndex)+nPanelLTopY+1,sData)

          break



        endSwitch
      break


    endSwitch

    if l_nKey!=-1 or !l_bFirst
      l_bFirst=true
      resize(sData,1,3)
      sData[0]="无"
      sData[1]="直线"
      sData[2]="圆弧"

      resize(sBuff,1,35)
      sBuff[0]="圆直径    :"+toString(".3",l_nData[0])
      sBuff[1]="圆弧度(焊):"+toString(".3",l_nData[1])

      sBuff[2]="X方向个数 :"+toString("",l_nData[2])
      sBuff[3]="X方向距离 :"+toString(".3",l_nData[3])
      sBuff[4]="Y方向个数 :"+toString("",l_nData[4])
      sBuff[5]="Y方向距离 :"+toString(".3",l_nData[5])

      sBuff[6]="引入类型  :"+sData[l_nData[6]]
      sBuff[7]="引入比例  :"+toString(".3",l_nData[7])
      sBuff[8]="引出类型  :"+sData[l_nData[8]]
      sBuff[9]="引出比例  :"+toString(".3",l_nData[9])



      sBuff[10]="坐标系X   :"+toString(".3",l_nData[10])
      sBuff[11]="坐标系Y   :"+toString(".3",l_nData[11])
      sBuff[12]="坐标系Z   :"+toString(".3",l_nData[12])
      sBuff[13]="坐标系RX  :"+toString(".3",l_nData[13])
      sBuff[14]="坐标系RY  :"+toString(".3",l_nData[14])
      sBuff[15]="坐标系RZ  :"+toString(".3",l_nData[15])


      sBuff[16]="路径偏差X :"+toString(".3",l_nData[16])
      sBuff[17]="路径偏差Y :"+toString(".3",l_nData[17])
      sBuff[18]="路径偏差Z :"+toString(".3",l_nData[18])
      sBuff[19]="路径偏差RX:"+toString(".3",l_nData[19])
      sBuff[20]="路径偏差RY:"+toString(".3",l_nData[20])
      sBuff[21]="路径偏差RZ:"+toString(".3",l_nData[21])


      sBuff[22]="七轴距离  :"+toString(".3",l_nData[22])
      sBuff[23]="七轴速度  :"+toString(".3",l_nData[23])
      sBuff[25]="激光开延时:"+toString(".3",l_nData[25])
      sBuff[26]="激光关延时:"+toString(".3",l_nData[26])
      sBuff[27]="边长1     :"+toString(".3",l_nData[27])
      sBuff[28]="边长2     :"+toString(".3",l_nData[28])
      sBuff[29]="收弧长(焊 :"+toString(".3",l_nData[29])
      resize(sData,1,2)
      //  sData[0]="内切"
      //  sData[1]="外切"
      //  sBuff[24]="类型      :"+sData[l_nData[24]]
      if !x_bWeld
        sData[0]="内切"
        sData[1]="外切"
        sBuff[24]="类型      :"+sData[l_nData[24]]
      else
        sData[0]="开"
        sData[1]="关"
        sBuff[24]="动作焊接  :"+sData[l_nData[24]]

      endIf
      //  sBuff[30]="穿孔工艺  :"+toString(".3",l_nData[30])
      //
      //
      if !x_bWeld
        sBuff[30]="穿孔工艺  :"+toString(".3",l_nData[30])
      else
        sBuff[30]="激光程序号:"+toString(".3",l_nData[30])
      endIf
      sBuff[31]="八轴距离  :"+toString(".3",l_nData[31])
      sBuff[32]="八轴速度  :"+toString(".3",l_nData[32])


      sBuff[33]="Z 个数(焊):"+toString("",l_nData[33])
      sBuff[34]="Z 距离(焊):"+toString(".3",l_nData[34])

      call Control_List(sBuff,l_nSelectIndex)

    endIf

  endWhile




end

--- Form_Action.pgx ---
public program Form_Action(string x_sTitle, string x_sPanelTitle, string& x_sList[], num& x_nSelectIndex, bool& x_bIO[], num x_nPresetIndex, string& x_sLable[])
  local num l_nNum
begin
  //为LasMAN3.6进行配置界面
 // cls()
  x_nSelectIndex=round(x_nSelectIndex)%500
  x_nPresetIndex=x_nPresetIndex%50
  title(x_sTitle)
   gotoxy(0,0)
  put("动作执行需上电!")
  gotoxy(0,2)
  put("动作参数:")





  call Control_PanelXY(22,0,15,10)
    for l_nNum=0 to size(x_sLable)-1
    gotoxy(0,l_nNum+3)
    put(left(x_sLable[l_nNum]+"                            ",nPanelLTopX-1))
    endFor
  call Control_Panel(x_sPanelTitle)
  setTextMode(sel(x_bIO[0],1,0))
  gotoxy(1,13)
  put("执行")

 setTextMode(0)

        gotoxy(21,13)
    put("上传")
    gotoxy(31,13)
    put("保存")

    gotoxy(26,13)
    put("修改")
    gotoxy(31,13)
    put("保存")

    gotoxy(36,13)
    put("退出")


  call Control_List(x_sList,x_nSelectIndex)



end

--- Form_Config.pgx ---
public program Form_Config(num& x_nNum[], num& x_nPointIndex)
  local string l_sBuff[2]
  local string l_sVersion
begin
  //为LasMAN3.6配置
  //主要是配置界面


  l_sBuff[0]="关"
  l_sBuff[1]="开"
  //轮询
  resize(sBuff,1,40)

  sBuff[0]="工具(Tool)X  :"+toString(".3",  x_nNum[0])
  sBuff[1]="工具(Tool)Y  :"+toString(".3",x_nNum[1])
  sBuff[2]="工具(Tool)Z  :"+toString(".3",x_nNum[2])
  sBuff[3]="工具(Tool)RX :"+toString(".3",x_nNum[3])
  sBuff[4]="工具(Tool)RY :"+toString(".3",x_nNum[4])
  sBuff[5]="工具(Tool)RZ :"+toString(".3",x_nNum[5])


  sBuff[6]="回零速度(m/min):"+toString(".3",x_nNum[6])
  sBuff[7]="不拆工具示教 :"+l_sBuff[x_nNum[7]]
  sBuff[8]="示教回退(启动:"+l_sBuff[x_nNum[8]]

  sBuff[9]="PWM频率高(HZ):"+toString(".3",x_nNum[9])
  sBuff[10]="PWM频率低(HZ):"+toString(".3",x_nNum[10])
  sBuff[11]="模拟量系数   :"+toString(".3",x_nNum[11])
  sBuff[12]="速度匹配(s)  :"+toString(".3",x_nNum[12])
  sBuff[13]="光斑补偿(mm) :"+toString(".3",x_nNum[13])


  sBuff[14]="开气延时(s)  :"+toString(".3",x_nNum[14])
  sBuff[15]="随动延时(s)  :"+toString(".3",x_nNum[15])
  sBuff[16]="工位延时(s)  :"+toString(".3",x_nNum[16])

  sBuff[17]="快捷速度(mm/s):"+toString("",x_nNum[17])
  sBuff[18]="快捷加速度(%):"+toString("",x_nNum[18])
  sBuff[19]="快捷Blend(mm):"+toString(".3",x_nNum[19])
  sBuff[20]="快捷工艺     :"+toString("",x_nNum[20])


  sBuff[21]="异步7轴(启动):"+l_sBuff[x_nNum[21]]
  sBuff[22]="7轴home点(mm):"+toString(".3",x_nNum[22])
  sBuff[23]="7轴安全点速度:"+toString(".3",x_nNum[23])
  sBuff[24]="7轴分度      :"+toString("",x_nNum[24])



  sBuff[25]="焊接(启动)   :"+l_sBuff[x_nNum[25]]
  sBuff[26]="焊接回退长度 :"+toString("",x_nNum[26])
  //sBuff[27]="步进(启动)   :"+l_sBuff[x_nNum[27]]
  sBuff[28]="步进距离(mm) :"+toString(".3",x_nNum[28])
  sBuff[29]="远程生产密码 :"+toString(".3",x_nNum[29])
  sBuff[30]="同工位多产品 :"+l_sBuff[x_nNum[30]]
  sBuff[27]="报警延时触发 :"+toString(".3",x_nNum[27])
  sBuff[31]="拐角速度自适 :"+l_sBuff[x_nNum[31]]


  sBuff[32]="异步8轴(启动):"+l_sBuff[x_nNum[32]]
  sBuff[33]="8轴home点(mm):"+toString(".3",x_nNum[33])
  sBuff[34]="8轴安全点速度:"+toString(".3",x_nNum[34])
  sBuff[35]="8轴分度      :"+toString("",x_nNum[35])

  sBuff[36]="工位完成IO输出:"+l_sBuff[x_nNum[36]]
  sBuff[37]="PLC控制外部轴:"+l_sBuff[x_nNum[37]]
  sBuff[38]="切割厚板模式 :"+l_sBuff[x_nNum[38]]


  call Control_LeftS(",,,,,上传,保存,退出,")
  call Control_PanelS("选项",17,0,20,10)
  call Control_BottomS(",,,,,上传,保存,退出,")
  call Control_List(sBuff,x_nPointIndex)


end

--- Form_Main.pgx ---
public program Form_Main(string& x_sBottomList[])
  local num l_nIndex
begin
  //欢迎界面，显示日期和时间
 userPage()
cls()
 call Control_PanelMd("下位机处在主界面")



//     for l_nIndex=0 to min(7,size(x_sBottomList)-1)
//    gotoxy(1+l_nIndex*5,13)
//    if size(x_sBottomList)>l_nIndex and x_sBottomList[l_nIndex]!=""
//      put(x_sBottomList[l_nIndex])
//    endIf
//    endFor
 call Control_Bottom(x_sBottomList)
end

--- Form_Product.pgx ---
public program Form_Product(string x_sTitle, string& x_sLableList[], string& x_sList[], string x_sBottom)
  local num l_nNum
begin

  //cls()
  title(x_sTitle)
  setTextMode(0)
  for l_nNum=0 to size(x_sLableList)-1
    gotoxy(0,l_nNum+1)
    if l_nNum==2
      setTextMode(2)
    endIf
    put(left(x_sLableList[l_nNum]+"            ",18))
    setTextMode(0)
    gotoxy(22,l_nNum+1)

    put(left(x_sList[l_nNum]+"            ",18))
  endFor

  //2016.03.07
  //为焊接修改
  if size(x_sList,1)==12 and x_sList[11]!=""
    gotoxy(22,12)
    put(left(x_sList[11]+"            ",17))
  endIf

  call Control_BottomS(x_sBottom)



end

--- Form_SelSharp.pgx ---
public program Form_SelSharp(num& x_nTypeIndex, bool& x_bRes)
  local string l_sList[13]
  local num l_nKey
  local num l_nIndex
begin
  //为LasMAN3.6
  //选择示教产品的类型


  l_nIndex=0
  l_sList[0]="不规则图形"
  l_sList[1]="圆-圆心直径法"
  l_sList[2]="圆-三点法"
  l_sList[3]="三角形"
  l_sList[4]="矩形"
  l_sList[5]="正五边形"
  l_sList[6]="正六边形"
  l_sList[7]="腰形"
  l_sList[8]="五角星(测)"
  l_sList[9]="圆管(测)"
  l_sList[10]="C形-三点法(焊)"
  l_sList[11]="同步不规则图形"
  l_sList[12]="同步空走路径"
  cls()

  //title(x_sTitle)

  call Control_PanelXY(0,0,15,10)
  call Control_Panel("图形类型")
  call Control_BottomS("示教,,,,,,,退出")

  //x_nSelectIndex=0
  call Control_List(l_sList,l_nIndex)

  while true
    l_nKey=getKey()
    switch l_nKey
      case 261
        l_nIndex=l_nIndex-1
        if l_nIndex<0
          l_nIndex=12
        endIf
        // l_nIndex=max(l_nIndex-1,0)
      break

      case 266
        l_nIndex=l_nIndex+1
        //l_nIndex=min(l_nIndex+1,11)

        if l_nIndex>12
          l_nIndex=0
        endIf


      break


      //示教,F1 和回车键
      case 271,270
        x_bRes=true
        switch l_nIndex
          case 0
            x_nTypeIndex=10
          break

          case 1
            x_nTypeIndex=2
          break

          case 2
            x_nTypeIndex=1
          break

          case 3
            x_nTypeIndex=3
          break

          case 4
            x_nTypeIndex=4
          break

          case 5
            x_nTypeIndex=5
          break

          case 6
            x_nTypeIndex=6
          break


          case 7
            x_nTypeIndex=7
          break



          case 8
            x_nTypeIndex=21
          break


          case 9
            x_nTypeIndex=22
          break


          case 10
            x_nTypeIndex=24
          break
          case 11
            x_nTypeIndex=20
          break

          case 12
            x_nTypeIndex=9
          break
        endSwitch

        return
      break

      //F8 和ESC键退出
      case 278,255
        x_bRes=false
        return

      break



    endSwitch

    if l_nKey!=-1

      call Control_List(l_sList,l_nIndex)
    endIf


  endWhile




end

--- Form_SimArray.pgx ---
public program Form_SimArray(string x_sTitle, string x_sPanelTitle, string& x_sList[], num& x_nSelectIndex, num& x_nPreset[], bool& x_bIO[], trsf x_trArray)
begin
  //为LasMAN3.6
  //工艺参数模拟选项


  //cls()
  x_nSelectIndex=round(x_nSelectIndex)%500

  title(x_sTitle)
  gotoxy(1,5)
  put("实时工艺参数:")
  x_trArray.x=sel(x_trArray.x==0,1,x_trArray.x)
  x_trArray.z=sel(x_trArray.z==0,1,x_trArray.z)
  x_trArray.ry=sel(x_trArray.ry==0,1,x_trArray.ry)


  if x_sPanelTitle=="切割点" or x_sPanelTitle=="工艺表"
    gotoxy(1,6)
    put("激光功率  :"+toString("",x_nPreset[0])+"   ")
    gotoxy(1,7)
    put("气体压力  :"+toString("",x_nPreset[3])+"   ")
    gotoxy(1,8)
    put("占空比频率:"+toString("",x_nPreset[1])+"   ")
    gotoxy(1,9)
    put("激光占空比:"+toString("",x_nPreset[2])+"   ")
    gotoxy(1,10)
    put("随动高度  :"+toString("",x_nPreset[4])+"   ")
    gotoxy(1,11)
    put("阵列:"+toString("",x_trArray.y)+"/"+toString("",x_trArray.x)+" "+toString("",x_trArray.rx)+"/"+toString("",x_trArray.z)+" "+toString("",x_trArray.rz)+"/"+toString("",x_trArray.ry)+" ")
  else
    gotoxy(1,6)
    put("激光功率  :0   ")
    gotoxy(1,7)
    put("气体压力  :0   ")
    gotoxy(1,8)
    put("占空比频率:0   ")
    gotoxy(1,9)
    put("激光占空比:0   ")
    gotoxy(1,10)
    put("随动高度  :0   ")

  endIf


  call Control_PanelXY(22,0,15,10)
  call Control_Panel(x_sPanelTitle)
  //call Control_BottomS("激光,随动,气体,,,,,终止")
  setTextMode(sel(x_bIO[0],1,0))
  gotoxy(1,13)
  put("激光")


  setTextMode(sel(x_bIO[1],1,0))
  gotoxy(6,13)
  put("随动")


  setTextMode(sel(x_bIO[2],01,0))
  gotoxy(11,13)
  put("气体")

  setTextMode(0)

  if  x_sPanelTitle=="工艺表"

    gotoxy(21,13)
    put("上传")

    gotoxy(26,13)
    put("修改")
    gotoxy(31,13)
    put("保存")

    gotoxy(36,13)
    put("退出")

  else
    gotoxy(36,13)
    put("终止")

  endIf
  //x_nSelectIndex=0
  call Control_List(x_sList,x_nSelectIndex)



end

--- Form_Simulation.pgx ---
public program Form_Simulation(string x_sTitle, string x_sPanelTitle, string& x_sList[], num& x_nSelectIndex, num& x_nPreset[], bool& x_bIO[])
begin
  //为LasMAN3.6
  //工艺参数模拟选项


  //cls()
  x_nSelectIndex=round(x_nSelectIndex)%500

  title(x_sTitle)
  gotoxy(1,5)
  put("实时工艺参数:")


  if x_sPanelTitle=="切割点" or x_sPanelTitle=="工艺表"
    gotoxy(1,6)
    put("激光功率  :"+toString("",x_nPreset[0])+"   ")
    gotoxy(1,7)
    put("气体压力  :"+toString("",x_nPreset[3])+"   ")
    gotoxy(1,8)
    put("占空比频率:"+toString("",x_nPreset[1])+"   ")
    gotoxy(1,9)
    put("激光占空比:"+toString("",x_nPreset[2])+"   ")
    gotoxy(1,10)
    put("随动高度  :"+toString("",x_nPreset[4])+"   ")
  else
    gotoxy(1,6)
    put("激光功率  :0   ")
    gotoxy(1,7)
    put("气体压力  :0   ")
    gotoxy(1,8)
    put("占空比频率:0   ")
    gotoxy(1,9)
    put("激光占空比:0   ")
    gotoxy(1,10)
    put("随动高度  :0   ")

  endIf


  call Control_PanelXY(22,0,15,10)
  call Control_Panel(x_sPanelTitle)
  //call Control_BottomS("激光,随动,气体,,,,,终止")
  setTextMode(sel(x_bIO[0],1,0))
  gotoxy(1,13)
  put("激光")


  setTextMode(sel(x_bIO[1],1,0))
  gotoxy(6,13)
  put("随动")


  setTextMode(sel(x_bIO[2],01,0))
  gotoxy(11,13)
  put("气体")

  setTextMode(0)

  if  x_sPanelTitle=="工艺表"

    gotoxy(21,13)
    put("上传")

    gotoxy(26,13)
    put("修改")
    gotoxy(31,13)
    put("保存")

    gotoxy(36,13)
    put("退出")

  else
    gotoxy(36,13)
    put("终止")

  endIf
  //x_nSelectIndex=0
  call Control_List(x_sList,x_nSelectIndex)



end

--- Int_EditMin.pgx ---
program Int_EditMin(num& x_nData, num x_nX, num x_nY, string x_sMess, num x_nMin)
  local num l_nKey
  local num l_nNum
  local num l_nOri
  local bool l_bBNum
begin
  //参数判断
  x_nX=min(max(0,x_nX),39)
  x_nY=min(max(0,x_nY),13)
  //x_nLength=min(max(1,x_nLength),39)

  //把字符串给打印出来
  gotoxy(x_nX,x_nY)
  setTextMode(0)
  put(x_sMess)

  //数值限定
  l_nNum=0
  for l_nKey=0 to nPanelWidthX-x_nX+nPanelLTopX+1-1
      l_nNum=l_nNum*10+9*l_nKey
  endFor

  l_nOri=x_nData
  l_bBNum=false
   l_nKey=0
  while l_nKey!=270 and l_nKey!=255
 //数值进行刷新，
 gotoxy(x_nX,x_nY)
 setTextMode(0)

 put(left("                ",nPanelWidthX-x_nX+nPanelLTopX+1-getDisplayLen(x_sMess)))


 //让其在编辑状态时 为白字黑底闪烁
   setTextMode(3)

//对按键进行判断
    l_nKey=getKey()
    switch l_nKey
      //从0～9进行编辑
      case 48,49,50,51,52,53,54,55,56,57
        if  !l_bBNum
          x_nData=0
          l_bBNum=true
        endIf
        if x_nData<l_nNum and x_nData>l_nNum*-1
          x_nData=x_nData*10+l_nKey-48
        endIf
      break


      //ESC
      case 255
        x_nData=l_nOri
        setTextMode(0)
      break
            //回车
      case 270
        setTextMode(0)
      break

      //UP
      case 261
        if !l_bBNum
          x_nData=x_nData+1
        endIf
      break
       //Down
      case 266
        if !l_bBNum
          x_nData=max(x_nData-1,x_nMin)
        endIf
      break

      //bp
      case 263
        l_bBNum=false
        x_nData=0
      break
    endSwitch
    x_nData=round(x_nData)



    //把数值给打印出来
    gotoxy(x_nX+getDisplayLen(x_sMess),x_nY)
    put(toString("",x_nData))
    delay(0)
  endWhile
end

--- Int_EditS.pgx ---
program Int_EditS(num& x_nData, num x_nX, num x_nY, string x_sMess)
  local num l_nKey
  local num l_nNum
  local num l_nOri
  local bool l_bBNum
begin

  call Int_EditMin(x_nData,x_nX,x_nY,x_sMess,0)
//  //参数判断
//  x_nX=min(max(0,x_nX),39)
//  x_nY=min(max(0,x_nY),13)
//  //x_nLength=min(max(1,x_nLength),39)
//
//  //把字符串给打印出来
//  gotoxy(x_nX,x_nY)
//  setTextMode(0)
//  put(x_sMess)
//
//  //数值限定
//  l_nNum=0
//  for l_nKey=0 to nPanelWidthX-x_nX+nPanelLTopX+1-1
//      l_nNum=l_nNum*10+9*l_nKey
//  endFor
//
//  l_nOri=x_nData
//  l_bBNum=false
//   l_nKey=0
//  while l_nKey!=270 and l_nKey!=255
// //数值进行刷新，
// gotoxy(x_nX,x_nY)
// setTextMode(0)
//
// put(left("                ",nPanelWidthX-x_nX+nPanelLTopX+1-getDisplayLen(x_sMess)))
//
//
// //让其在编辑状态时 为白字黑底闪烁
//   setTextMode(3)
//
////对按键进行判断
//    l_nKey=getKey()
//    switch l_nKey
//      //从0～9进行编辑
//      case 48,49,50,51,52,53,54,55,56,57
//        if  !l_bBNum
//          x_nData=0
//          l_bBNum=true
//        endIf
//        if x_nData<l_nNum and x_nData>l_nNum*-1
//          x_nData=x_nData*10+l_nKey-48
//        endIf
//      break
//
//
//      //ESC
//      case 255
//        x_nData=l_nOri
//        setTextMode(0)
//      break
//            //回车
//      case 270
//        setTextMode(0)
//      break
//
//      //UP
//      case 261
//        if !l_bBNum
//          x_nData=x_nData+1
//        endIf
//      break
//       //Down
//      case 266
//        if !l_bBNum
//          x_nData=max(x_nData-1,0)
//        endIf
//      break
//
//      //bp
//      case 263
//        l_bBNum=false
//        x_nData=0
//      break
//    endSwitch
//    x_nData=round(x_nData)
//
//
//
//    //把数值给打印出来
//    gotoxy(x_nX+getDisplayLen(x_sMess),x_nY)
//    put(toString("",x_nData))
//    delay(0)
//  endWhile
end
